// Mitsubishi GX Works2 project: DMOV   PLC: Q02/Q02H

PROGRAM MAIN
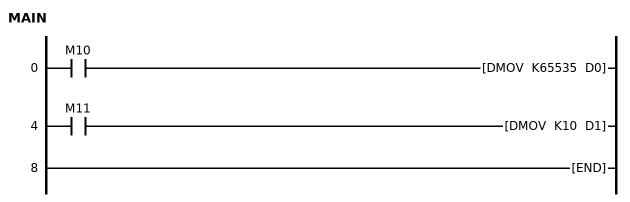
0     LD      M10
      DMOV    K65535 D0
4     LD      M11
      DMOV    K10 D1
8     END
END_PROGRAM
